Fanuc KAREL source: kt00712.KL

-- PROVISIONAL review KL for V940-1; original PC SHA256 c154163d03343b8cb8e120917292f5918624bda6e2dcaddeb0f00d149cc9d077
-- Incomplete behavior may be omitted. Consult companion uncertainty JSON. Do not deploy.
PROGRAM KT00712
%NOLOCKGROUP
VAR
  S1 : STRING[80]
  S2 : STRING[80]
  OUT : BOOLEAN
BEGIN
  -- V9_ZERO_TABLE_METADATA_HINT layout=0001; no indexed target words; source/name/runtime held
  -- UNRESOLVED_PC offsets 5-14; opcodes 3F,75
  -- UNRESOLVED_PC offsets 19-28; opcodes 3F,75
  -- UNRESOLVED_PC offsets 33-42; opcodes 3F,75
  -- UNRESOLVED_PC offsets 47-56; opcodes 3F,75
  -- UNRESOLVED_PC offsets 61-76; opcodes 22,63,23
  -- UNRESOLVED_PC offsets 81-85; opcodes 7F
END KT00712
